# EPICS substitutions: db/Beckhoff_1XXX/ecmcEK1501-0010.substitutions
file "ecmcEcSlave.template"
{
  pattern {}
          {}
}

file "ecmc_coupler-ID.template"
{
  pattern {}
          {}
}
